// TIA Portal V17 export
// export: Created 2022-04-06T07:28:40.0356852Z, ExportSetting WithDefaults, DisplayName Totally Integrated Automation Portal, DisplayVersion V17, DisplayName TIA Portal Openness, DisplayVersion V17, DisplayName TIA Portal Version Control Interface, DisplayVersion V17, DisplayName TIA Portal Test Suite Advanced, DisplayVersion V17, DisplayName SINAMICS Startdrive Advanced, DisplayVersion V17, DisplayName SINAMICS Startdrive G130, G150, S120, S150, SINAMICS MV, S210, DisplayVersion V17, DisplayName SINAMICS Startdrive G110M, G120, G120C, G120D, G120P, G115D, DisplayVersion V17, DisplayName STEP 7 Professional, DisplayVersion V17, DisplayName STEP 7 Safety, DisplayVersion V17, DisplayName WinCC Advanced / Unified PC, DisplayVersion V17
DATA_BLOCK "InstFileHandling"   // DB15
VERSION : 0.1
// stored: AutoNumber true, DBAccessibleFromOPCUA true, DBAccessibleFromWebserver true, InstanceOfName FileHandling, InstanceOfType FB
"FileHandling"
   // VAR
   //    instFileWriteC_SFB { S7_SetPoint := 'True'} : FileWriteC;
   //    instFileReadC_SFB { S7_SetPoint := 'True'} : FileReadC;
   //    instFileDelete { S7_SetPoint := 'True'} : FileDelete;
   //    statData { S7_SetPoint := 'True'} : Array[0..3] of Byte;
   // END_VAR
BEGIN
END_DATA_BLOCK
